// TIA Portal V19 export
FUNCTION_BLOCK "Pu_CM05.GP11"   // FB1011, LAD
TITLE = Pumpe GP11: Entleeren CM05
{ S7_Optimized_Access := 'TRUE' }
// Funktionen:  Entleeren /  Spülen
// stored: AutoNumber false, MemoryReserve 100, SetENOAutomatically false
   VAR RETAIN
      In { ExternalVisible := 'False'; ExternalWritable := 'False'} : Struct
         NotHalt : Bool;
         MSS_ok : Bool;
         Auto : Bool;   // Paneltaste
         Ein : Bool;   // Paneltaste
         GW_p : Bool;
         "Niv_Uel_CM05.BL05" : Bool;
         "Niv_max_CM05.BL01" : Bool;
         "Niv_min_CM05.BL02" : Bool;
         "Niv_TLS_CM05.BL03" : Bool;
         AWA_ok : Bool;
         Frg_AWA : Bool;
         "SRM_CM05.QM61_auf" : Bool;
         "SRM_CM05.QM61_zu" : Bool;
         "SRM_CM05.QM64_auf" : Bool;
         "SRM_CM05.QM64_zu" : Bool;
         Betriebsart : USInt := 0;   // Paneltaste
         Druck_Pumpe { ExternalAccessible := 'False'} : Real;
      END_STRUCT;
      Param { ExternalVisible := 'False'; ExternalWritable := 'False'} : Struct
         Spülzeit : Time;
         DT_Druckaufbau { ExternalAccessible := 'False'} : Time;
         DT_Testzeit { ExternalAccessible := 'False'} : Time;
         SW_Drucktest { ExternalAccessible := 'False'} : Real;
      END_STRUCT;
      Zst : Struct
         Niveau : USInt;
         Status_GP11 : USInt;
         Status_DT { ExternalAccessible := 'False'; ExternalVisible := 'False'; ExternalWritable := 'False'} : USInt;
         Restzeit_Spülen : Time;
         Restzeit_DT { ExternalAccessible := 'False'; ExternalVisible := 'False'; ExternalWritable := 'False'} : Time;
         "TON_CM05.QM62_auf" : Bool;
         Spuelen : Bool;
         Zeit_laeuft { ExternalAccessible := 'False'; ExternalVisible := 'False'; ExternalWritable := 'False'} : Bool;
         Spuelen_aktiv : Bool;
         Drucktest_aktiv : Bool;
         Drucktest_ok { ExternalAccessible := 'False'; ExternalVisible := 'False'; ExternalWritable := 'False'} : Bool;
         Bedienung_erlaubt { ExternalAccessible := 'False'; ExternalVisible := 'False'; ExternalWritable := 'False'} : Bool;
      END_STRUCT;
      Mld { ExternalVisible := 'False'; ExternalWritable := 'False'} : Struct
         MSS : Bool;
         "TLS_CM05.BL03" : Bool;
         "Uel_CM05.BL05" : Bool;
         AWA_niO : Bool;
         keine_Frg_AWA : Bool;
         Niv_Sensorfehler : Bool;
         GW_p : Bool;
         n_Auto : Bool;
         TO_Druckaufbau { ExternalAccessible := 'False'} : Bool;
         Drucktest_ok { ExternalAccessible := 'False'} : Bool;
         DT_Fehler { ExternalAccessible := 'False'} : Bool;
         Pu_Spuelen_Fertig { ExternalAccessible := 'False'} : Bool;
      END_STRUCT;
      Out { ExternalVisible := 'False'; ExternalWritable := 'False'} : Struct
         GP11_Ein : Bool;
         QM61 : Bool;
         QM62 : Bool;
         QM63 : Bool;
         QM64 : Bool;
      END_STRUCT;
   END_VAR
   VAR
      IEC_Timer : Struct
         "CM05.QM62_auf" { ExternalAccessible := 'False'; ExternalVisible := 'False'; ExternalWritable := 'False'; S7_SetPoint := 'True'} : TON_TIME;
         Spülen { S7_SetPoint := 'True'} : TP_TIME;
         GW_p { S7_SetPoint := 'True'} : TON_TIME;
         Drucktest { ExternalAccessible := 'False'; ExternalVisible := 'False'; ExternalWritable := 'False'; S7_SetPoint := 'True'} : TP_TIME;
         TO_Druckaufbau { ExternalAccessible := 'False'; ExternalVisible := 'False'; ExternalWritable := 'False'; S7_SetPoint := 'True'} : TON_TIME;
         QM63 { S7_SetPoint := 'True'} : TOF_TIME;
      END_STRUCT;
      R_TRIG_Hand_EIN { S7_SetPoint := 'True'} : R_TRIG;
   END_VAR
   VAR_TEMP
      Spülzeit : Time;
      Zeit_DT : Time;
      GP11_Laeuft : Bool;
      posFl_Hand : Bool;
   END_VAR
   VAR CONSTANT
      Niv_TLS : USInt := 7;
      Niv_Min : USInt := 35;
      Niv_max : USInt := 85;
      Niv_Uel : USInt := 98;
      Zeit_Ventil_auf : Time := T#3s;
      S1 : USInt := 1;
      S2 : USInt := 2;
      S3 : USInt := 3;
      S4 : USInt := 4;
      "Name" : String := 'Pu CM05.GP11';
   END_VAR
BEGIN

REGION Network 1 (SCL): Input
   // Panelbedienung und Sensoren --> Input()
   // Not-Halt
   #In.NotHalt := NOT "DB_PNOZ_IN_Out".In.NH_Frg_Pumpen;
   // Timer Spülventil AUF
   #IEC_Timer."CM05.QM62_auf"(IN := #Out.QM62,
                              PT := #Zeit_Ventil_auf,
                              Q => #Zst."TON_CM05.QM62_auf");
   // positive Flanke "Hand Ein"
   #R_TRIG_Hand_EIN(CLK := #In.Ein,
                    Q => #posFl_Hand);
END_REGION

REGION Network 2 (SCL): Pumpe Ein Entleerung Sammeltank CM05.GP11
   IF #In.MSS_ok AND NOT #In.NotHalt THEN

       // "Normal"-Betrieb
       #Zst.Bedienung_erlaubt := NOT #In.Ein AND NOT #In.Auto AND NOT #Mld.DT_Fehler;

       //Drucktest rücksetzen
       IF #In.Betriebsart <> 2 OR #Zst.Spuelen_aktiv OR NOT #In.Ein THEN
           #Mld.Drucktest_ok := FALSE;
           #Mld.DT_Fehler := FALSE;
           #Mld.TO_Druckaufbau := FALSE;
           #Zst.Status_DT := 0;
           #Zst.Drucktest_aktiv := FALSE;
       END_IF;
       //Spülmeldung rücksetzen
       IF #In.Betriebsart <> 1 OR NOT #In.Ein THEN
           #Mld.Pu_Spuelen_Fertig := FALSE;
       END_IF;

       CASE #In.Betriebsart OF
           0:  // Entleeren
               #Out.QM64 := #In.AWA_ok AND #In.Frg_AWA;
               // Spülventile zu
               #Out.QM62 := FALSE;
               #Out.QM63 := FALSE;
               #Zst.Restzeit_Spülen := T#0s;
               #Zst.Drucktest_aktiv := FAlSE;

               // Zwischen MAX und MIN entleeren oder einmalig per Hand
               IF (#In.Auto AND #In."Niv_max_CM05.BL01" OR #posFl_Hand ) AND #In."Niv_TLS_CM05.BL03"THEN
                   #Out.QM61 := TRUE;
               ELSIF NOT #In."Niv_TLS_CM05.BL03" OR NOT #In."Niv_min_CM05.BL02" OR (NOT #In.Auto AND NOT #In.Ein) THEN
                       #Out.QM61 := FALSE;
                END_IF;

               //Pumpe an, wenn Ventile geöffnet sind
                #Out.GP11_Ein := #In."SRM_CM05.QM61_auf" AND #In."SRM_CM05.QM64_auf" AND #In."Niv_TLS_CM05.BL03";

            1: // Spülen - nur Hand
                // Ventile Abpumpen zu    
                #Out.QM61 := FALSE;
                #Out.QM64 := FALSE;

                // Ausschaltverzögert - Druckabbau
                #IEC_Timer.QM63(IN := #Out.QM62,
                                PT := T#3s,
                                Q => #Out.QM63);

                IF #In.Ein THEN
                        IF #posFl_Hand THEN
                            #Zst.Spuelen_aktiv := TRUE;
                        END_IF;
                        #Out.QM62 := NOT #In."Niv_max_CM05.BL01" AND #In."SRM_CM05.QM61_zu" AND #In."SRM_CM05.QM64_zu" AND NOT #In."Niv_Uel_CM05.BL05" AND #Zst.Spuelen_aktiv;

                        #IEC_Timer.Spülen(IN := #Zst."TON_CM05.QM62_auf" AND #Out.QM63,
                                          PT := #Param.Spülzeit,
                                          Q => #Zst.Spuelen,
                                          ET => #Spülzeit);
                        #Zst.Restzeit_Spülen := #Param.Spülzeit - #Spülzeit;

                        IF #Zst."TON_CM05.QM62_auf" AND #Out.QM63 AND #In."SRM_CM05.QM61_zu" AND #In."SRM_CM05.QM64_zu" AND NOT #Zst.Spuelen THEN
                            #Zst.Spuelen_aktiv := FALSE;
                            #Out.QM62 := FALSE;
                        END_IF;

                        // Fertig
                        IF NOT #Zst.Spuelen AND NOT #Zst.Spuelen_aktiv AND NOT #Out.QM63 THEN
                            #Out.QM62 := #Out.QM63 := FALSE;
                            #Zst.Restzeit_Spülen := T#0s;
                            #Mld.Pu_Spuelen_Fertig := TRUE;
                        END_IF;
                    ELSE
                        #Out.QM62 := FALSE;
                        #Out.QM63 := FALSE;
                        #Zst.Restzeit_Spülen := T#0s;
                    END_IF;
                    #Out.GP11_Ein := FALSE;

           2: // Spülen + Drucktest - nur Hand
               // Ventile Abpumpen zu    
               #Out.QM61 := FALSE;
               #Out.QM64 := FALSE;
               IF NOT #Zst.Drucktest_aktiv THEN
                   IF #In.Ein THEN
                       IF #posFl_Hand THEN
                           #Zst.Spuelen_aktiv := TRUE;
                       END_IF;
                       #Out.QM62 := NOT #In."Niv_max_CM05.BL01" AND NOT #In."Niv_Uel_CM05.BL05";
                       #Out.QM63 := #Out.QM62;
                       #IEC_Timer.Spülen(IN := #Zst."TON_CM05.QM62_auf" AND #Out.QM63 AND #In."SRM_CM05.QM61_zu" AND #In."SRM_CM05.QM64_zu",
                                         PT := #Param.Spülzeit,
                                         Q => #Zst.Spuelen,
                                         ET => #Spülzeit);
                       #Zst.Restzeit_Spülen := #Param.Spülzeit - #Spülzeit;

                       IF #Zst."TON_CM05.QM62_auf" AND #Out.QM63 AND #In."SRM_CM05.QM61_zu" AND #In."SRM_CM05.QM64_zu" AND NOT #Zst.Spuelen THEN
                           #Zst.Spuelen_aktiv := FALSE;
                       END_IF;

                       // Fertig
                       IF NOT #Zst.Spuelen AND NOT #Zst.Spuelen_aktiv THEN
                           #Out.QM62 := #Out.QM63 := FALSE;
                           #Zst.Restzeit_Spülen := T#0s;
                           #Zst.Drucktest_aktiv := TRUE;
                           #Zst.Status_DT := #S1;
                       END_IF;
                   ELSE
                       #Out.QM62 := FALSE;
                       #Out.QM63 := FALSE;
                       #Zst.Restzeit_Spülen := T#0s;
                   END_IF;
                   #Out.GP11_Ein := FALSE;
               END_IF;

               IF #Zst.Drucktest_aktiv THEN
                   CASE #Zst.Status_DT OF
                       #S1:  //Druckaufbau

                           IF "DB_Temporaer".Drucksensoren_deaktiviert THEN
                               #Zst.Drucktest_ok := TRUE;

                               "Ergebnis_DT"("Name" := #"Name",
                                             akt_Zeit := "Uhrzeit".aktDatum,
                                             ok := #Zst.Drucktest_ok,
                                             Fehler := NOT #Zst.Drucktest_ok);

                               #Mld.Drucktest_ok := #Zst.Drucktest_ok;
                               #Mld.DT_Fehler := NOT #Zst.Drucktest_ok;
                               #Zst.Status_DT := #S4;
                           ELSE
                               #Out.QM62 := TRUE;
                               IF (#In.Druck_Pumpe > #Param.SW_Drucktest + 0.25) OR #Mld.TO_Druckaufbau THEN
                                   #Zst.Status_DT := #S2;
                               END_IF;
                               #Zst.Restzeit_DT := #Param.DT_Druckaufbau - #IEC_Timer.TO_Druckaufbau.ET;
                           END_IF;

                       #S2: //Wartezeit
                           #IEC_Timer.Drucktest(IN := NOT #Out.QM62,
                                                PT := #Param.DT_Testzeit,
                                                Q => #Zst.Zeit_laeuft,
                                                ET => #Zeit_DT);
                           #Zst.Restzeit_DT := #Param.DT_Testzeit - #Zeit_DT;

                           IF NOT #Zst.Zeit_laeuft AND NOT #Out.QM62 THEN
                               #Zst.Restzeit_DT := T#0s;
                               #Zst.Status_DT := #S3;
                           END_IF;
                           #Out.QM62 := FALSE;

                       #S3:// Überprüfung
                           #Zst.Drucktest_ok := #In.Druck_Pumpe >= #Param.SW_Drucktest;

                           "Ergebnis_DT"("Name" := #"Name",
                                         akt_Zeit := "Uhrzeit".aktDatum,
                                         ok := #Zst.Drucktest_ok,
                                         Fehler := NOT #Zst.Drucktest_ok);

                           #Mld.Drucktest_ok := #Zst.Drucktest_ok;
                           #Mld.DT_Fehler := NOT #Zst.Drucktest_ok;
                           #Zst.Status_DT := #S4;

                       #S4: // Ende
                           ;
                   END_CASE;
               END_IF;
       END_CASE;
   ELSE
       #Out.GP11_Ein := FALSE;
       #Out.QM61 := FALSE;
       #Out.QM62 := FALSE;
       #Out.QM63 := FALSE;
       #Out.QM64 := FALSE;
   END_IF;
END_REGION

REGION Network 3 (SCL): Überwachung / Meldungen
   // Motorschutzschalter
   #Mld.MSS := NOT #In.MSS_ok AND NOT #In.NotHalt;
   // Trockenlaufschutz
   #Mld."TLS_CM05.BL03" := NOT #In."Niv_TLS_CM05.BL03";
   // Überlauf
   #Mld."Uel_CM05.BL05" := #In."Niv_Uel_CM05.BL05";
   // AWA nicht betriebsbereit
   #Mld.AWA_niO := NOT #In.AWA_ok;
   // keine Freigabe Abpumpen
   #Mld.keine_Frg_AWA := NOT #In.Frg_AWA;

   // Zeitüberschreitung Druckaufbau
   #IEC_Timer.TO_Druckaufbau(IN := #Zst.Status_DT = #S1,
                             PT := #Param.DT_Druckaufbau,
                             Q => #Mld.TO_Druckaufbau);

   // Grenzwert Pumpendruck
   #IEC_Timer.GW_p(IN := #Out.GP11_Ein,
                   PT := T#3s,
                   Q => #GP11_Laeuft);

   #Mld.GW_p := #GP11_Laeuft AND #In.GW_p;
   // nicht in Automatik
   #Mld.n_Auto := NOT #In.Auto AND "DB_ANLAGE".BA.Automat_ein;
END_REGION

REGION Network 4 (SCL): --> Visu
   // Status Pumpe
   "Status_E0A"(Hand := #In.Ein,
                Auto := #In.Auto,
                SonderModus_PumpeSpuelen:=#Zst.Spuelen,
                Stoerung := NOT #In.MSS_ok,
                Ausgang := #Out.GP11_Ein,
                StatusByte => #Zst.Status_GP11);
   // Anzeige Füllstand
   "Niv_Visu"(Niv_1 := #In."Niv_TLS_CM05.BL03",
              Niv_2 := #In."Niv_min_CM05.BL02",
              Niv_3 := #In."Niv_max_CM05.BL01",
              Niv_4 := #In."Niv_Uel_CM05.BL05",
              Niv_5 := FALSE,
              Niv_6 := FALSE,
              Wert_1 := #Niv_TLS,
              Wert_2 := #Niv_Min,
              Wert_3 := #Niv_max,
              Wert_4 := #Niv_Uel,
              Wert_5 := 0,
              Wert_6 := 0,
              Niveau => #Zst.Niveau,
              Niv_Err => #Mld.Niv_Sensorfehler);
END_REGION
END_FUNCTION_BLOCK
